PROGRAM TestAlarmFB
VAR
	arrFbAlarm : ARRAY[1..10] OF FB_HandleAlarms;
	arrbRaiseAlarm:	ARRAY[1..10] OF BOOL;
	bClearAllAlarms:BOOL;
	index:USINT;
	index2:USINT;
END_VAR

clearAllAlarms();

mapAlarmTexts();

setEventClass();

raiseAlarms();

mapEvents();

mapSourceName();

ACTION clearAllAlarms:
//clear all alarms
IF bClearAllAlarms THEN
	FOR index:=1 TO 10 DO 
		arrFbAlarm[index].ClearAlarm();
	END_FOR
	
	IF index=10 THEN
		bClearAllAlarms:=0;
	END_IF
END_IF
END_ACTION

ACTION mapAlarmTexts:

FOR index:=1 TO 10 DO 
	arrFbAlarm[index].sEventClass:='AlarmSystem';
END_FOR
END_ACTION

ACTION mapEvents:
//map alarm texts
arrFbAlarm[1].sEvent:='Alarm1';
arrFbAlarm[2].sEvent:='Alarm2';
arrFbAlarm[3].sEvent:='Alarm3';
arrFbAlarm[4].sEvent:='Alarm4';
arrFbAlarm[5].sEvent:='Alarm5';
arrFbAlarm[6].sEvent:='Alarm6';
arrFbAlarm[7].sEvent:='Alarm7';
arrFbAlarm[8].sEvent:='Alarm8';
arrFbAlarm[9].sEvent:='Alarm9';
arrFbAlarm[10].sEvent:='Alarm10';
END_ACTION

ACTION mapSourceName:
//map alarm texts
arrFbAlarm[1].sSourceName:='Source 1';
arrFbAlarm[2].sSourceName:='Source 2';
arrFbAlarm[3].sSourceName:='Source 3';
arrFbAlarm[4].sSourceName:='Source 4';
arrFbAlarm[5].sSourceName:='Source 5';
arrFbAlarm[6].sSourceName:='Source 6';
arrFbAlarm[7].sSourceName:='Source 7';
arrFbAlarm[8].sSourceName:='Source 8';
arrFbAlarm[8].sSourceName:='Source 9';
arrFbAlarm[10].sSourceName:='Source 10';
END_ACTION

ACTION raiseAlarms:
IF arrbRaiseAlarm[1] THEN 
	arrFbAlarm[1].RaiseAlarm();
END_IF

IF arrbRaiseAlarm[2] THEN 
	arrFbAlarm[2].RaiseAlarm();
END_IF


IF arrbRaiseAlarm[3] THEN 
	arrFbAlarm[3].RaiseAlarm();
END_IF

IF arrbRaiseAlarm[4] THEN 
	arrFbAlarm[4].RaiseAlarm();
END_IF

IF arrbRaiseAlarm[5] THEN 
	arrFbAlarm[5].RaiseAlarm();
END_IF

IF arrbRaiseAlarm[6] THEN 
	arrFbAlarm[6].RaiseAlarm();
END_IF

IF arrbRaiseAlarm[7] THEN 
	arrFbAlarm[7].RaiseAlarm();
END_IF

IF arrbRaiseAlarm[8] THEN 
	arrFbAlarm[8].RaiseAlarm();
END_IF

IF arrbRaiseAlarm[9] THEN 
	arrFbAlarm[9].RaiseAlarm();
END_IF

IF arrbRaiseAlarm[10] THEN 
	arrFbAlarm[10].RaiseAlarm();
END_IF
END_ACTION

ACTION setEventClass:

//map alarm texts
arrFbAlarm[1].sAlarmText:='Alarm 1';
arrFbAlarm[2].sAlarmText:='Alarm 2';
arrFbAlarm[3].sAlarmText:='Alarm 3';
arrFbAlarm[4].sAlarmText:='Alarm 4';
arrFbAlarm[5].sAlarmText:='Alarm 5';
arrFbAlarm[6].sAlarmText:='Alarm 6';
arrFbAlarm[7].sAlarmText:='Alarm 7';
arrFbAlarm[8].sAlarmText:='Alarm 8';
arrFbAlarm[9].sAlarmText:='Alarm 9';
arrFbAlarm[10].sAlarmText:='Alarm 10';
END_ACTION

END_PROGRAM

(* stored: Version 1.1.0.1, ProductVersion 3.1.4024.11
   POU TestAlarmFB: Id {faa7c60d-2ac0-409a-98f2-ab8518de51bd}, SpecialFunc None
   Action clearAllAlarms: Id {26c7d649-505b-4a40-a428-7d1224000042}
   Action mapAlarmTexts: Id {a2bc7ecb-fb0e-442c-8530-15623a4c0e12}
   Action mapEvents: Id {afefe776-dc76-46ff-9e31-4104b86e2cde}
   Action mapSourceName: Id {5d57aed9-8c83-4f59-9bb7-96581da15f06}
   Action raiseAlarms: Id {06ed3250-47aa-4867-a5dd-fb15d340b8aa}
   Action setEventClass: Id {2c43a8a8-10f5-4cef-b64b-af73d3b18252} *)
